W52.14 BOOL  ; 腔体下料#2夹爪气缸松开复位(M)
W52.15 BOOL  ; 腔体下料#3夹爪气缸夹紧复位(M)
W57.00 BOOL  ; 进料移栽有料信号
W60.00 BOOL  ; 腔体机构手复位
W60.01 BOOL  ; 腔体#1 & #2复位启动
W60.02 BOOL  ; 腔体#3 & #4复位启动
W61.01 BOOL  ; #1抽真空阀复位
W61.02 BOOL  ; #2抽真空阀复位
W61.03 BOOL  ; #1氦检阀复位
W61.04 BOOL  ; #2氦检阀复位
W61.05 BOOL  ; #1总氦检阀复位
W61.07 BOOL  ; #1合模气缸缩回位复位
W61.09 BOOL  ; #2合模气缸缩回位复位
W61.11 BOOL  ; 破真空阀#1&#2复位
W61.12 BOOL  ; 关破真空阀#1&#2复位
W61.15 BOOL  ; #1 & #2吹气阀复位
W62.00 BOOL  ; #2吹气阀复位
W62.01 BOOL  ; #3 & #4吹气阀复位
W62.03 BOOL  ; #3抽真空阀复位
W62.04 BOOL  ; #4抽真空阀复位
W62.06 BOOL  ; #2总氦检阀复位
W62.07 BOOL  ; 破真空阀#3&#4复位
W62.08 BOOL  ; 关破真空阀#3&#4复位
W62.09 BOOL  ; #3氦检阀复位
W62.10 BOOL  ; #4氦检阀复位
W62.11 BOOL  ; #3合模气缸缩回位复位
W62.12 BOOL  ; 破真空阀#3&#4复位
W62.13 BOOL  ; #4合模气缸缩回位复位
W70.00 BOOL  ; 出料机构手复位
W9.00 BOOL  ; 故障
W9.01 BOOL  ; 报警清除  HMI

## Program Main (cyclic task 0)
Local symbols
P_on BOOL

### Section 启停控制

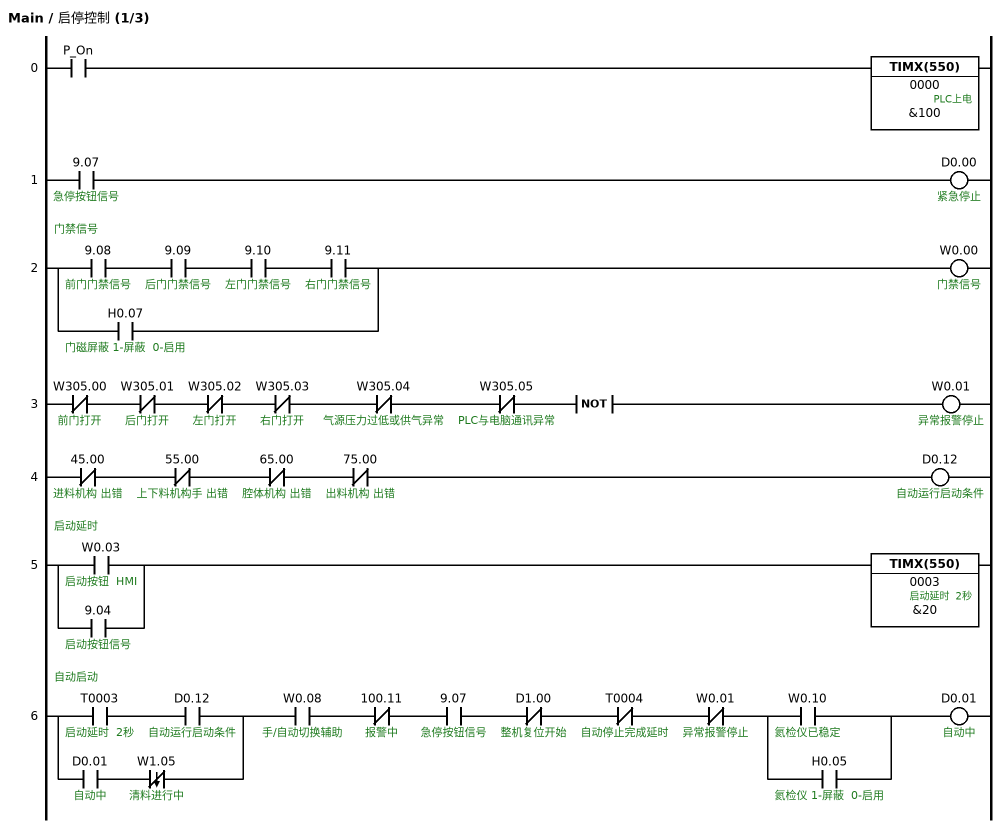
; rung 0
LD P_On
TIMX(550) 0000 &100  ; PLC上电
; rung 1
LD 9.07  ; 急停按钮信号
OUT D0.00  ; 紧急停止
; rung 2: 门禁信号
LD 9.08  ; 前门门禁信号
AND 9.09  ; 后门门禁信号
AND 9.10  ; 左门门禁信号
AND 9.11  ; 右门门禁信号
OR H0.07  ; 门磁屏蔽 1-屏蔽  0-启用
OUT W0.00  ; 门禁信号
; rung 3
LDNOT W305.00  ; 前门打开
ANDNOT W305.01  ; 后门打开
ANDNOT W305.02  ; 左门打开
ANDNOT W305.03  ; 右门打开
ANDNOT W305.04  ; 气源压力过低或供气异常
ANDNOT W305.05  ; PLC与电脑通讯异常
NOT(520)
OUT W0.01  ; 异常报警停止
; rung 4
LDNOT 45.00  ; 进料机构 出错
ANDNOT 55.00  ; 上下料机构手 出错
ANDNOT 65.00  ; 腔体机构 出错
ANDNOT 75.00  ; 出料机构 出错
OUT D0.12  ; 自动运行启动条件
; rung 5: 启动延时
LD W0.03  ; 启动按钮  HMI
OR 9.04  ; 启动按钮信号
TIMX(550) 0003 &20  ; 启动延时  2秒
; rung 6: 自动启动
LD T0003  ; 启动延时  2秒
AND D0.12  ; 自动运行启动条件
LD D0.01  ; 自动中
%ANDNOT W1.05  ; 清料进行中
ORLD
AND W0.08  ; 手/自动切换辅助
ANDNOT 100.11  ; 报警中
AND 9.07  ; 急停按钮信号
ANDNOT D1.00  ; 整机复位开始
ANDNOT T0004  ; 自动停止完成延时
ANDNOT W0.01  ; 异常报警停止
LD W0.10  ; 氦检仪已稳定
OR H0.05  ; 氦检仪 1-屏蔽  0-启用
ANDLD
OUT D0.01  ; 自动中

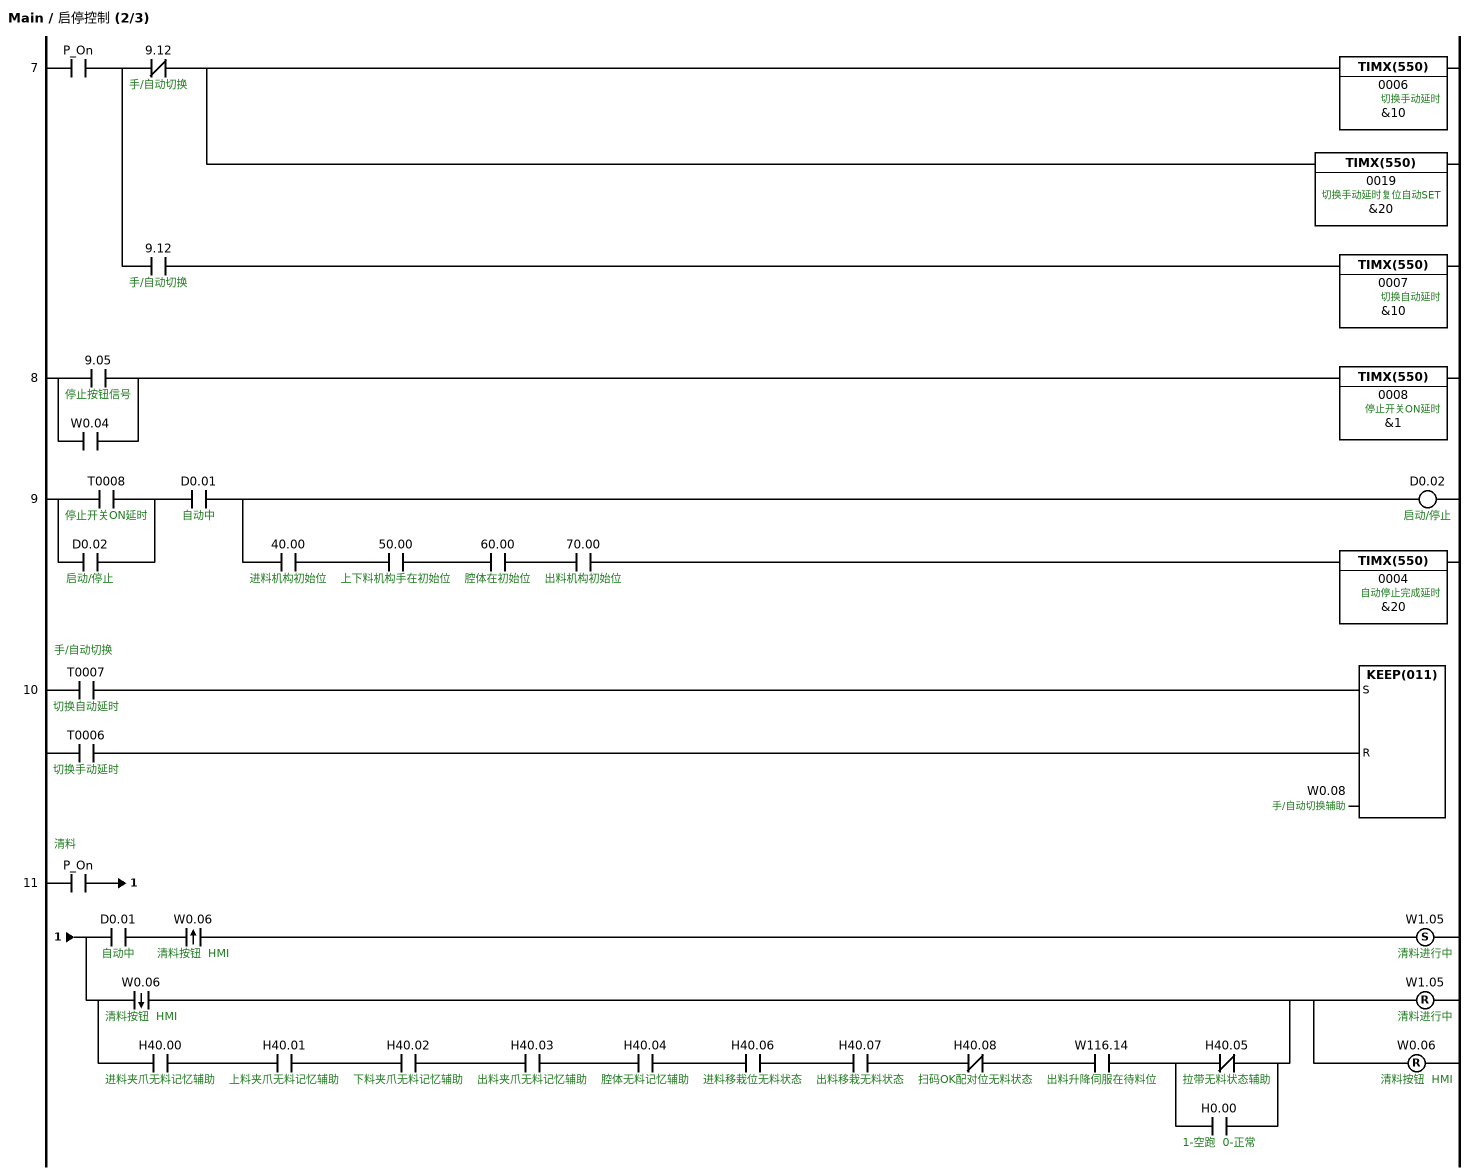
; rung 7
LD P_On
OUT TR0
ANDNOT 9.12  ; 手/自动切换
TIMX(550) 0006 &10  ; 切换手动延时
TIMX(550) 0019 &20  ; 切换手动延时复位自动SET
LD TR0
AND 9.12  ; 手/自动切换
TIMX(550) 0007 &10  ; 切换自动延时
; rung 8
LD 9.05  ; 停止按钮信号
OR W0.04
TIMX(550) 0008 &1  ; 停止开关ON延时
; rung 9
LD T0008  ; 停止开关ON延时
OR D0.02  ; 启动/停止
AND D0.01  ; 自动中
OUT D0.02  ; 启动/停止
AND 40.00  ; 进料机构初始位
AND 50.00  ; 上下料机构手在初始位
AND 60.00  ; 腔体在初始位
AND 70.00  ; 出料机构初始位
TIMX(550) 0004 &20  ; 自动停止完成延时
; rung 10: 手/自动切换
LD T0007  ; 切换自动延时
LD T0006  ; 切换手动延时
KEEP(011) W0.08  ; 手/自动切换辅助
; rung 11: 清料
LD P_On
OUT TR0
AND D0.01  ; 自动中
@AND W0.06  ; 清料按钮  HMI
SET W1.05  ; 清料进行中
LD TR0
%LD W0.06  ; 清料按钮  HMI
LD H40.00  ; 进料夹爪无料记忆辅助
AND H40.01  ; 上料夹爪无料记忆辅助
AND H40.02  ; 下料夹爪无料记忆辅助
AND H40.03  ; 出料夹爪无料记忆辅助
AND H40.04  ; 腔体无料记忆辅助
AND H40.06  ; 进料移栽位无料状态
AND H40.07  ; 出料移栽无料状态
ANDNOT H40.08  ; 扫码OK配对位无料状态
AND W116.14  ; 出料升降伺服在待料位
LDNOT H40.05  ; 拉带无料状态辅助
OR H0.00  ; 1-空跑  0-正常
ANDLD
ORLD
ANDLD
RSET W1.05  ; 清料进行中
RSET W0.06  ; 清料按钮  HMI

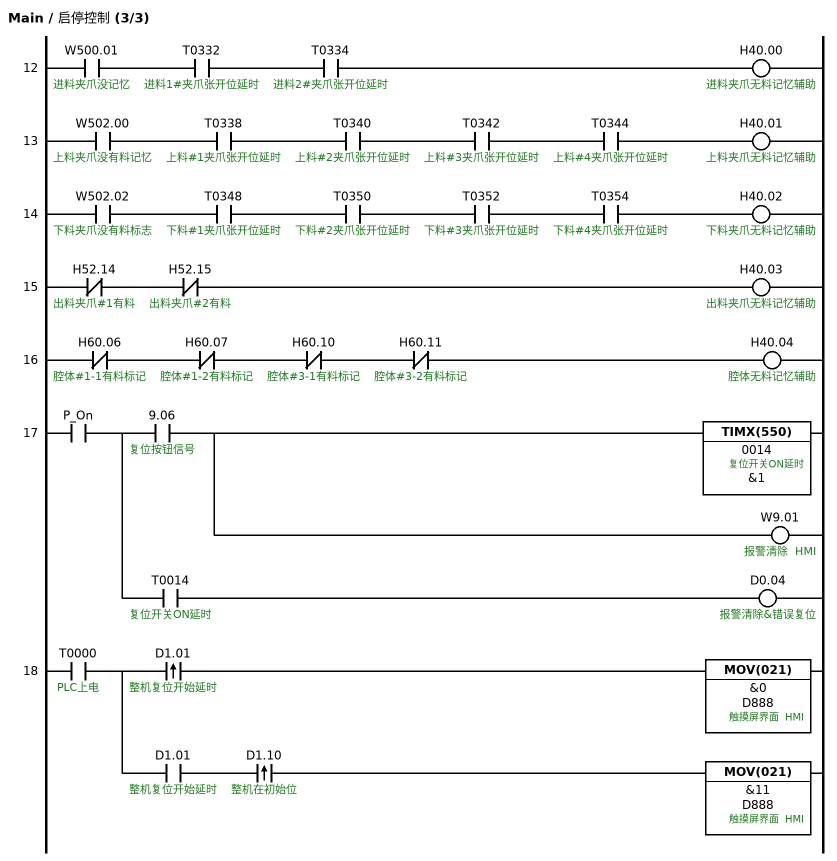
; rung 12
LD W500.01  ; 进料夹爪没记忆
AND T0332  ; 进料1#夹爪张开位延时
AND T0334  ; 进料2#夹爪张开位延时
OUT H40.00  ; 进料夹爪无料记忆辅助
; rung 13
LD W502.00  ; 上料夹爪没有料记忆
AND T0338  ; 上料#1夹爪张开位延时
AND T0340  ; 上料#2夹爪张开位延时
AND T0342  ; 上料#3夹爪张开位延时
AND T0344  ; 上料#4夹爪张开位延时
OUT H40.01  ; 上料夹爪无料记忆辅助
; rung 14
LD W502.02  ; 下料夹爪没有料标志
AND T0348  ; 下料#1夹爪张开位延时
AND T0350  ; 下料#2夹爪张开位延时
AND T0352  ; 下料#3夹爪张开位延时
AND T0354  ; 下料#4夹爪张开位延时
OUT H40.02  ; 下料夹爪无料记忆辅助
; rung 15
LDNOT H52.14  ; 出料夹爪#1有料
ANDNOT H52.15  ; 出料夹爪#2有料
OUT H40.03  ; 出料夹爪无料记忆辅助
; rung 16
LDNOT H60.06  ; 腔体#1-1有料标记
ANDNOT H60.07  ; 腔体#1-2有料标记
ANDNOT H60.10  ; 腔体#3-1有料标记
ANDNOT H60.11  ; 腔体#3-2有料标记
OUT H40.04  ; 腔体无料记忆辅助
; rung 17
LD P_On
OUT TR0
AND 9.06  ; 复位按钮信号
TIMX(550) 0014 &1  ; 复位开关ON延时
OUT W9.01  ; 报警清除  HMI
LD TR0
AND T0014  ; 复位开关ON延时
OUT D0.04  ; 报警清除&错误复位
; rung 18
LD T0000  ; PLC上电
OUT TR0
@AND D1.01  ; 整机复位开始延时
MOV(021) &0 D888  ; 触摸屏界面  HMI
LD TR0
AND D1.01  ; 整机复位开始延时
@AND D1.10  ; 整机在初始位
MOV(021) &11 D888  ; 触摸屏界面  HMI

### Section 传感器延时及屏蔽

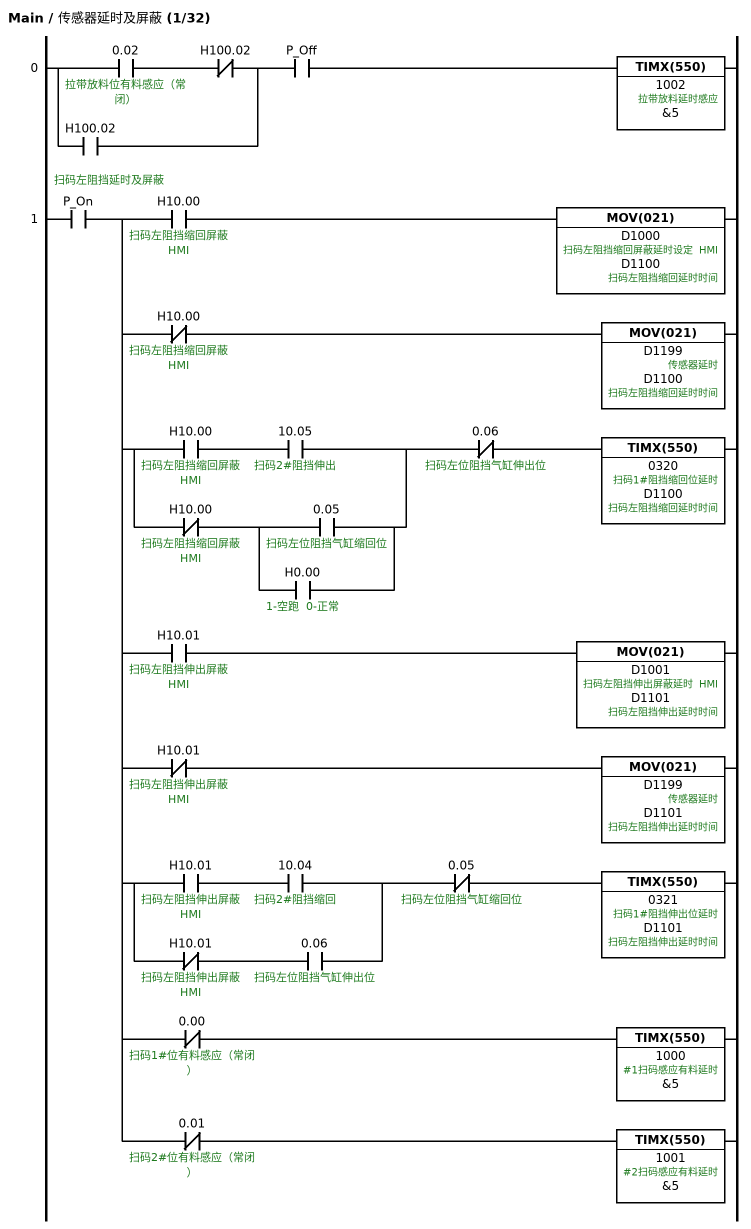
; rung 0
LD 0.02  ; 拉带放料位有料感应（常闭）
ANDNOT H100.02
OR H100.02
AND P_Off
TIMX(550) 1002 &5  ; 拉带放料延时感应
; rung 1: 扫码左阻挡延时及屏蔽
LD P_On
OUT TR0
AND H10.00  ; 扫码左阻挡缩回屏蔽  HMI
MOV(021) D1000 D1100  ; 扫码左阻挡缩回屏蔽延时设定  HMI, 扫码左阻挡缩回延时时间
LD TR0
ANDNOT H10.00  ; 扫码左阻挡缩回屏蔽  HMI
MOV(021) D1199 D1100  ; 传感器延时, 扫码左阻挡缩回延时时间
LD TR0
LD H10.00  ; 扫码左阻挡缩回屏蔽  HMI
AND 10.05  ; 扫码2#阻挡伸出
LDNOT H10.00  ; 扫码左阻挡缩回屏蔽  HMI
LD 0.05  ; 扫码左位阻挡气缸缩回位
OR H0.00  ; 1-空跑  0-正常
ANDLD
ORLD
ANDLD
ANDNOT 0.06  ; 扫码左位阻挡气缸伸出位
TIMX(550) 0320 D1100  ; 扫码左阻挡缩回延时时间, 扫码1#阻挡缩回位延时
LD TR0
AND H10.01  ; 扫码左阻挡伸出屏蔽  HMI
MOV(021) D1001 D1101  ; 扫码左阻挡伸出屏蔽延时  HMI, 扫码左阻挡伸出延时时间
LD TR0
ANDNOT H10.01  ; 扫码左阻挡伸出屏蔽  HMI
MOV(021) D1199 D1101  ; 传感器延时, 扫码左阻挡伸出延时时间
LD TR0
LD H10.01  ; 扫码左阻挡伸出屏蔽  HMI
AND 10.04  ; 扫码2#阻挡缩回
LDNOT H10.01  ; 扫码左阻挡伸出屏蔽  HMI
AND 0.06  ; 扫码左位阻挡气缸伸出位
ORLD
ANDLD
ANDNOT 0.05  ; 扫码左位阻挡气缸缩回位
TIMX(550) 0321 D1101  ; 扫码左阻挡伸出延时时间, 扫码1#阻挡伸出位延时
LD TR0
ANDNOT 0.00  ; 扫码1#位有料感应（常闭）
TIMX(550) 1000 &5  ; #1扫码感应有料延时
LD TR0
ANDNOT 0.01  ; 扫码2#位有料感应（常闭）
TIMX(550) 1001 &5  ; #2扫码感应有料延时

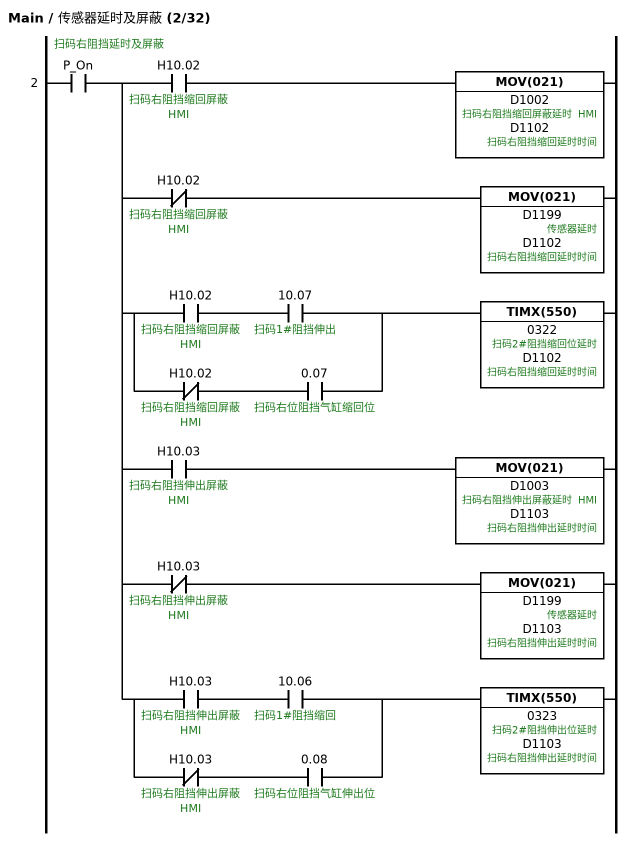
; rung 2: 扫码右阻挡延时及屏蔽
LD P_On
OUT TR0
AND H10.02  ; 扫码右阻挡缩回屏蔽  HMI
MOV(021) D1002 D1102  ; 扫码右阻挡缩回屏蔽延时  HMI, 扫码右阻挡缩回延时时间
LD TR0
ANDNOT H10.02  ; 扫码右阻挡缩回屏蔽  HMI
MOV(021) D1199 D1102  ; 传感器延时, 扫码右阻挡缩回延时时间
LD TR0
LD H10.02  ; 扫码右阻挡缩回屏蔽  HMI
AND 10.07  ; 扫码1#阻挡伸出
LDNOT H10.02  ; 扫码右阻挡缩回屏蔽  HMI
AND 0.07  ; 扫码右位阻挡气缸缩回位
ORLD
ANDLD
TIMX(550) 0322 D1102  ; 扫码右阻挡缩回延时时间, 扫码2#阻挡缩回位延时
LD TR0
AND H10.03  ; 扫码右阻挡伸出屏蔽  HMI
MOV(021) D1003 D1103  ; 扫码右阻挡伸出屏蔽延时  HMI, 扫码右阻挡伸出延时时间
LD TR0
ANDNOT H10.03  ; 扫码右阻挡伸出屏蔽  HMI
MOV(021) D1199 D1103  ; 传感器延时, 扫码右阻挡伸出延时时间
LD TR0
LD H10.03  ; 扫码右阻挡伸出屏蔽  HMI
AND 10.06  ; 扫码1#阻挡缩回
LDNOT H10.03  ; 扫码右阻挡伸出屏蔽  HMI
AND 0.08  ; 扫码右位阻挡气缸伸出位
ORLD
ANDLD
TIMX(550) 0323 D1103  ; 扫码右阻挡伸出延时时间, 扫码2#阻挡伸出位延时

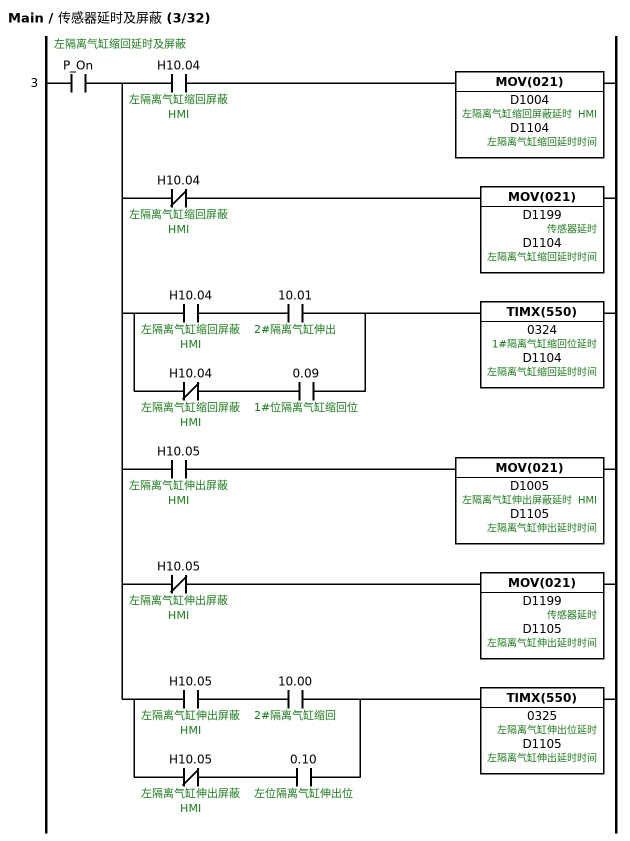
; rung 3: 左隔离气缸缩回延时及屏蔽
LD P_On
OUT TR0
AND H10.04  ; 左隔离气缸缩回屏蔽  HMI
MOV(021) D1004 D1104  ; 左隔离气缸缩回屏蔽延时  HMI, 左隔离气缸缩回延时时间
LD TR0
ANDNOT H10.04  ; 左隔离气缸缩回屏蔽  HMI
MOV(021) D1199 D1104  ; 传感器延时, 左隔离气缸缩回延时时间
LD TR0
LD H10.04  ; 左隔离气缸缩回屏蔽  HMI
AND 10.01  ; 2#隔离气缸伸出
LDNOT H10.04  ; 左隔离气缸缩回屏蔽  HMI
AND 0.09  ; 1#位隔离气缸缩回位
ORLD
ANDLD
TIMX(550) 0324 D1104  ; 左隔离气缸缩回延时时间, 1#隔离气缸缩回位延时
LD TR0
AND H10.05  ; 左隔离气缸伸出屏蔽  HMI
MOV(021) D1005 D1105  ; 左隔离气缸伸出屏蔽延时  HMI, 左隔离气缸伸出延时时间
LD TR0
ANDNOT H10.05  ; 左隔离气缸伸出屏蔽  HMI
MOV(021) D1199 D1105  ; 传感器延时, 左隔离气缸伸出延时时间
LD TR0
LD H10.05  ; 左隔离气缸伸出屏蔽  HMI
AND 10.00  ; 2#隔离气缸缩回
LDNOT H10.05  ; 左隔离气缸伸出屏蔽  HMI
AND 0.10  ; 左位隔离气缸伸出位
ORLD
ANDLD
TIMX(550) 0325 D1105  ; 左隔离气缸伸出延时时间, 左隔离气缸伸出位延时

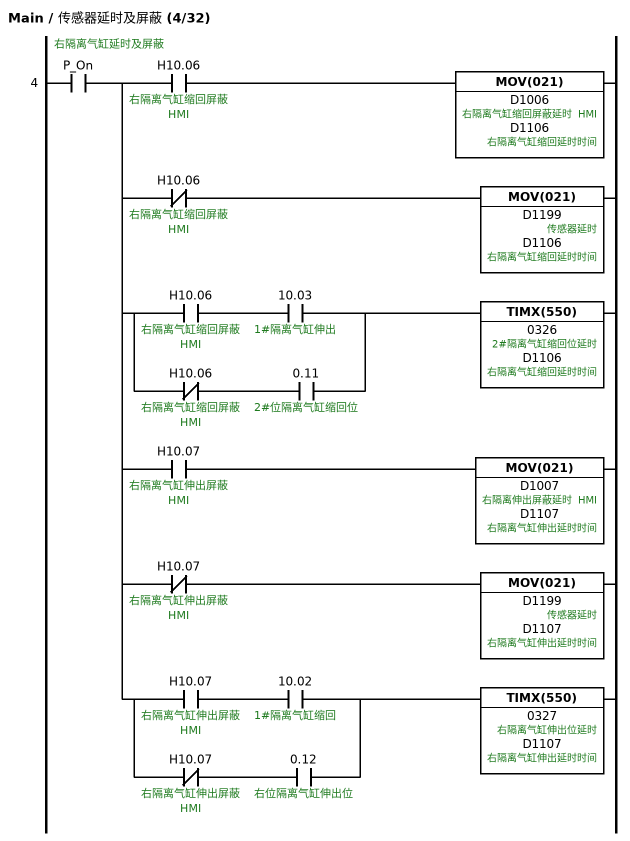
; rung 4: 右隔离气缸延时及屏蔽
LD P_On
OUT TR0
AND H10.06  ; 右隔离气缸缩回屏蔽  HMI
MOV(021) D1006 D1106  ; 右隔离气缸缩回屏蔽延时  HMI, 右隔离气缸缩回延时时间
LD TR0
ANDNOT H10.06  ; 右隔离气缸缩回屏蔽  HMI
MOV(021) D1199 D1106  ; 传感器延时, 右隔离气缸缩回延时时间
LD TR0
LD H10.06  ; 右隔离气缸缩回屏蔽  HMI
AND 10.03  ; 1#隔离气缸伸出
LDNOT H10.06  ; 右隔离气缸缩回屏蔽  HMI
AND 0.11  ; 2#位隔离气缸缩回位
ORLD
ANDLD
TIMX(550) 0326 D1106  ; 右隔离气缸缩回延时时间, 2#隔离气缸缩回位延时
LD TR0
AND H10.07  ; 右隔离气缸伸出屏蔽  HMI
MOV(021) D1007 D1107  ; 右隔离伸出屏蔽延时  HMI, 右隔离气缸伸出延时时间
LD TR0
ANDNOT H10.07  ; 右隔离气缸伸出屏蔽  HMI
MOV(021) D1199 D1107  ; 传感器延时, 右隔离气缸伸出延时时间
LD TR0
LD H10.07  ; 右隔离气缸伸出屏蔽  HMI
AND 10.02  ; 1#隔离气缸缩回
LDNOT H10.07  ; 右隔离气缸伸出屏蔽  HMI
AND 0.12  ; 右位隔离气缸伸出位
ORLD
ANDLD
TIMX(550) 0327 D1107  ; 右隔离气缸伸出延时时间, 右隔离气缸伸出位延时

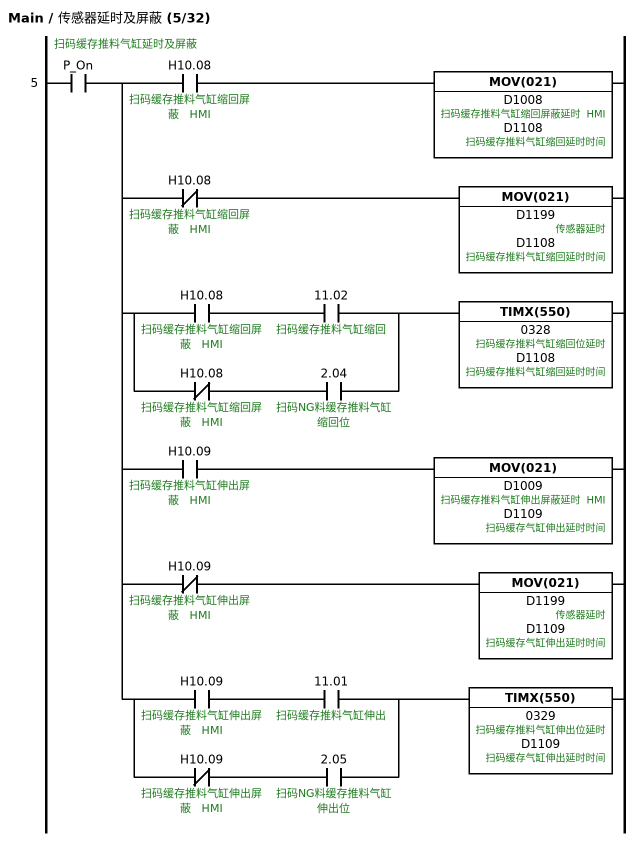
; rung 5: 扫码缓存推料气缸延时及屏蔽
LD P_On
OUT TR0
AND H10.08  ; 扫码缓存推料气缸缩回屏蔽   HMI
MOV(021) D1008 D1108  ; 扫码缓存推料气缸缩回屏蔽延时  HMI, 扫码缓存推料气缸缩回延时时间
LD TR0
ANDNOT H10.08  ; 扫码缓存推料气缸缩回屏蔽   HMI
MOV(021) D1199 D1108  ; 传感器延时, 扫码缓存推料气缸缩回延时时间
LD TR0
LD H10.08  ; 扫码缓存推料气缸缩回屏蔽   HMI
AND 11.02  ; 扫码缓存推料气缸缩回
LDNOT H10.08  ; 扫码缓存推料气缸缩回屏蔽   HMI
AND 2.04  ; 扫码NG料缓存推料气缸缩回位
ORLD
ANDLD
TIMX(550) 0328 D1108  ; 扫码缓存推料气缸缩回延时时间, 扫码缓存推料气缸缩回位延时
LD TR0
AND H10.09  ; 扫码缓存推料气缸伸出屏蔽   HMI
MOV(021) D1009 D1109  ; 扫码缓存推料气缸伸出屏蔽延时  HMI, 扫码缓存气缸伸出延时时间
LD TR0
ANDNOT H10.09  ; 扫码缓存推料气缸伸出屏蔽   HMI
MOV(021) D1199 D1109  ; 传感器延时, 扫码缓存气缸伸出延时时间
LD TR0
LD H10.09  ; 扫码缓存推料气缸伸出屏蔽   HMI
AND 11.01  ; 扫码缓存推料气缸伸出
LDNOT H10.09  ; 扫码缓存推料气缸伸出屏蔽   HMI
AND 2.05  ; 扫码NG料缓存推料气缸伸出位
ORLD
ANDLD
TIMX(550) 0329 D1109  ; 扫码缓存气缸伸出延时时间, 扫码缓存推料气缸伸出位延时

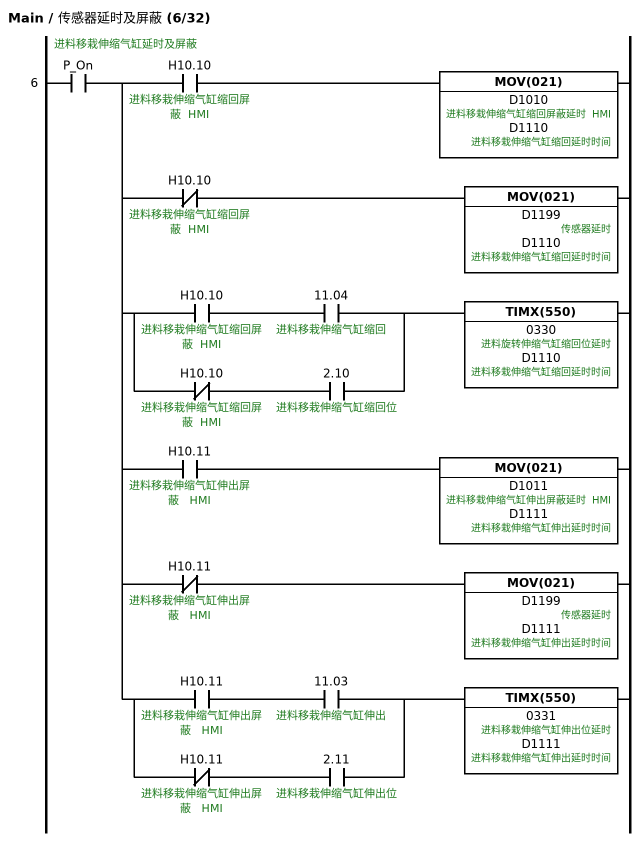
; rung 6: 进料移栽伸缩气缸延时及屏蔽
LD P_On
OUT TR0
AND H10.10  ; 进料移栽伸缩气缸缩回屏蔽  HMI
MOV(021) D1010 D1110  ; 进料移栽伸缩气缸缩回屏蔽延时  HMI, 进料移栽伸缩气缸缩回延时时间
LD TR0
ANDNOT H10.10  ; 进料移栽伸缩气缸缩回屏蔽  HMI
MOV(021) D1199 D1110  ; 传感器延时, 进料移栽伸缩气缸缩回延时时间
LD TR0
LD H10.10  ; 进料移栽伸缩气缸缩回屏蔽  HMI
AND 11.04  ; 进料移栽伸缩气缸缩回
LDNOT H10.10  ; 进料移栽伸缩气缸缩回屏蔽  HMI
AND 2.10  ; 进料移栽伸缩气缸缩回位
ORLD
ANDLD
TIMX(550) 0330 D1110  ; 进料移栽伸缩气缸缩回延时时间, 进料旋转伸缩气缸缩回位延时
LD TR0
AND H10.11  ; 进料移栽伸缩气缸伸出屏蔽   HMI
MOV(021) D1011 D1111  ; 进料移栽伸缩气缸伸出屏蔽延时  HMI, 进料移栽伸缩气缸伸出延时时间
LD TR0
ANDNOT H10.11  ; 进料移栽伸缩气缸伸出屏蔽   HMI
MOV(021) D1199 D1111  ; 传感器延时, 进料移栽伸缩气缸伸出延时时间
LD TR0
LD H10.11  ; 进料移栽伸缩气缸伸出屏蔽   HMI
AND 11.03  ; 进料移栽伸缩气缸伸出
LDNOT H10.11  ; 进料移栽伸缩气缸伸出屏蔽   HMI
AND 2.11  ; 进料移栽伸缩气缸伸出位
ORLD
ANDLD
TIMX(550) 0331 D1111  ; 进料移栽伸缩气缸伸出延时时间, 进料移栽伸缩气缸伸出位延时

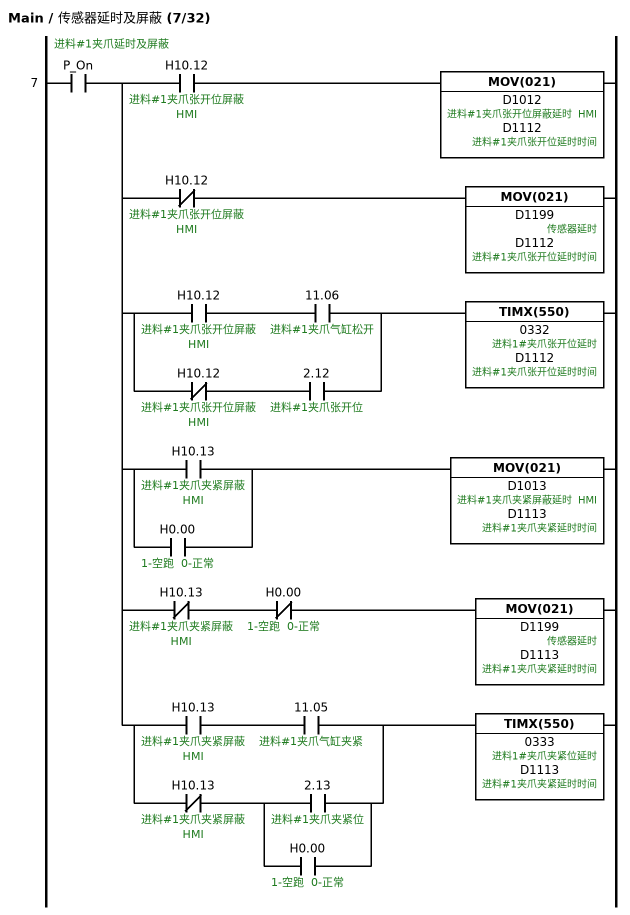
; rung 7: 进料#1夹爪延时及屏蔽
LD P_On
OUT TR0
AND H10.12  ; 进料#1夹爪张开位屏蔽  HMI
MOV(021) D1012 D1112  ; 进料#1夹爪张开位屏蔽延时  HMI, 进料#1夹爪张开位延时时间
LD TR0
ANDNOT H10.12  ; 进料#1夹爪张开位屏蔽  HMI
MOV(021) D1199 D1112  ; 传感器延时, 进料#1夹爪张开位延时时间
LD TR0
LD H10.12  ; 进料#1夹爪张开位屏蔽  HMI
AND 11.06  ; 进料#1夹爪气缸松开
LDNOT H10.12  ; 进料#1夹爪张开位屏蔽  HMI
AND 2.12  ; 进料#1夹爪张开位
ORLD
ANDLD
TIMX(550) 0332 D1112  ; 进料#1夹爪张开位延时时间, 进料1#夹爪张开位延时
LD TR0
LD H10.13  ; 进料#1夹爪夹紧屏蔽  HMI
OR H0.00  ; 1-空跑  0-正常
ANDLD
MOV(021) D1013 D1113  ; 进料#1夹爪夹紧屏蔽延时  HMI, 进料#1夹爪夹紧延时时间
LD TR0
ANDNOT H10.13  ; 进料#1夹爪夹紧屏蔽  HMI
ANDNOT H0.00  ; 1-空跑  0-正常
MOV(021) D1199 D1113  ; 传感器延时, 进料#1夹爪夹紧延时时间
LD TR0
LD H10.13  ; 进料#1夹爪夹紧屏蔽  HMI
AND 11.05  ; 进料#1夹爪气缸夹紧
LDNOT H10.13  ; 进料#1夹爪夹紧屏蔽  HMI
LD 2.13  ; 进料#1夹爪夹紧位
OR H0.00  ; 1-空跑  0-正常
ANDLD
ORLD
ANDLD
TIMX(550) 0333 D1113  ; 进料#1夹爪夹紧延时时间, 进料1#夹爪夹紧位延时

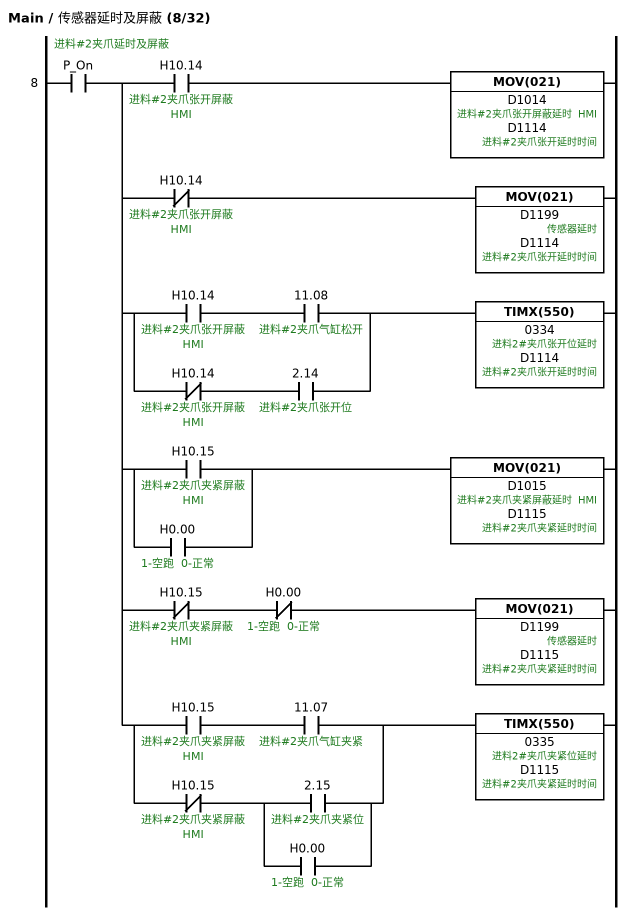
; rung 8: 进料#2夹爪延时及屏蔽
LD P_On
OUT TR0
AND H10.14  ; 进料#2夹爪张开屏蔽  HMI
MOV(021) D1014 D1114  ; 进料#2夹爪张开屏蔽延时  HMI, 进料#2夹爪张开延时时间
LD TR0
ANDNOT H10.14  ; 进料#2夹爪张开屏蔽  HMI
MOV(021) D1199 D1114  ; 传感器延时, 进料#2夹爪张开延时时间
LD TR0
LD H10.14  ; 进料#2夹爪张开屏蔽  HMI
AND 11.08  ; 进料#2夹爪气缸松开
LDNOT H10.14  ; 进料#2夹爪张开屏蔽  HMI
AND 2.14  ; 进料#2夹爪张开位
ORLD
ANDLD
TIMX(550) 0334 D1114  ; 进料#2夹爪张开延时时间, 进料2#夹爪张开位延时
LD TR0
LD H10.15  ; 进料#2夹爪夹紧屏蔽  HMI
OR H0.00  ; 1-空跑  0-正常
ANDLD
MOV(021) D1015 D1115  ; 进料#2夹爪夹紧屏蔽延时  HMI, 进料#2夹爪夹紧延时时间
LD TR0
ANDNOT H10.15  ; 进料#2夹爪夹紧屏蔽  HMI
ANDNOT H0.00  ; 1-空跑  0-正常
MOV(021) D1199 D1115  ; 传感器延时, 进料#2夹爪夹紧延时时间
LD TR0
LD H10.15  ; 进料#2夹爪夹紧屏蔽  HMI
AND 11.07  ; 进料#2夹爪气缸夹紧
LDNOT H10.15  ; 进料#2夹爪夹紧屏蔽  HMI
LD 2.15  ; 进料#2夹爪夹紧位
OR H0.00  ; 1-空跑  0-正常
ANDLD
ORLD
ANDLD
TIMX(550) 0335 D1115  ; 进料#2夹爪夹紧延时时间, 进料2#夹爪夹紧位延时

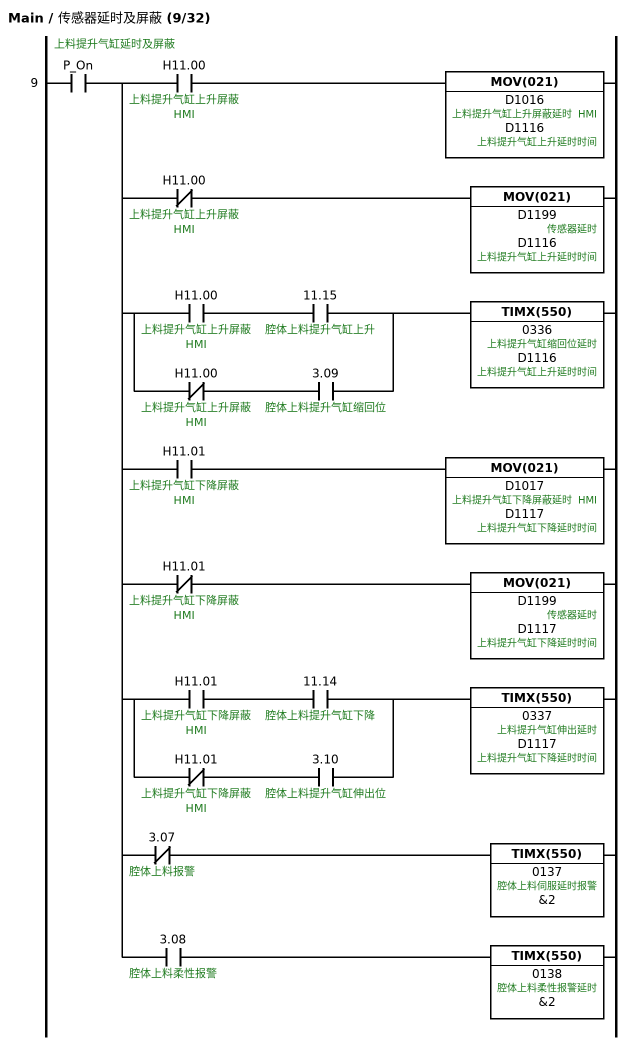
; rung 9: 上料提升气缸延时及屏蔽
LD P_On
OUT TR0
AND H11.00  ; 上料提升气缸上升屏蔽  HMI
MOV(021) D1016 D1116  ; 上料提升气缸上升屏蔽延时  HMI, 上料提升气缸上升延时时间
LD TR0
ANDNOT H11.00  ; 上料提升气缸上升屏蔽  HMI
MOV(021) D1199 D1116  ; 传感器延时, 上料提升气缸上升延时时间
LD TR0
LD H11.00  ; 上料提升气缸上升屏蔽  HMI
AND 11.15  ; 腔体上料提升气缸上升
LDNOT H11.00  ; 上料提升气缸上升屏蔽  HMI
AND 3.09  ; 腔体上料提升气缸缩回位
ORLD
ANDLD
TIMX(550) 0336 D1116  ; 上料提升气缸上升延时时间, 上料提升气缸缩回位延时
LD TR0
AND H11.01  ; 上料提升气缸下降屏蔽  HMI
MOV(021) D1017 D1117  ; 上料提升气缸下降屏蔽延时  HMI, 上料提升气缸下降延时时间
LD TR0
ANDNOT H11.01  ; 上料提升气缸下降屏蔽  HMI
MOV(021) D1199 D1117  ; 传感器延时, 上料提升气缸下降延时时间
LD TR0
LD H11.01  ; 上料提升气缸下降屏蔽  HMI
AND 11.14  ; 腔体上料提升气缸下降
LDNOT H11.01  ; 上料提升气缸下降屏蔽  HMI
AND 3.10  ; 腔体上料提升气缸伸出位
ORLD
ANDLD
TIMX(550) 0337 D1117  ; 上料提升气缸下降延时时间, 上料提升气缸伸出延时
LD TR0
ANDNOT 3.07  ; 腔体上料报警
TIMX(550) 0137 &2  ; 腔体上料伺服延时报警
LD TR0
AND 3.08  ; 腔体上料柔性报警
TIMX(550) 0138 &2  ; 腔体上料柔性报警延时

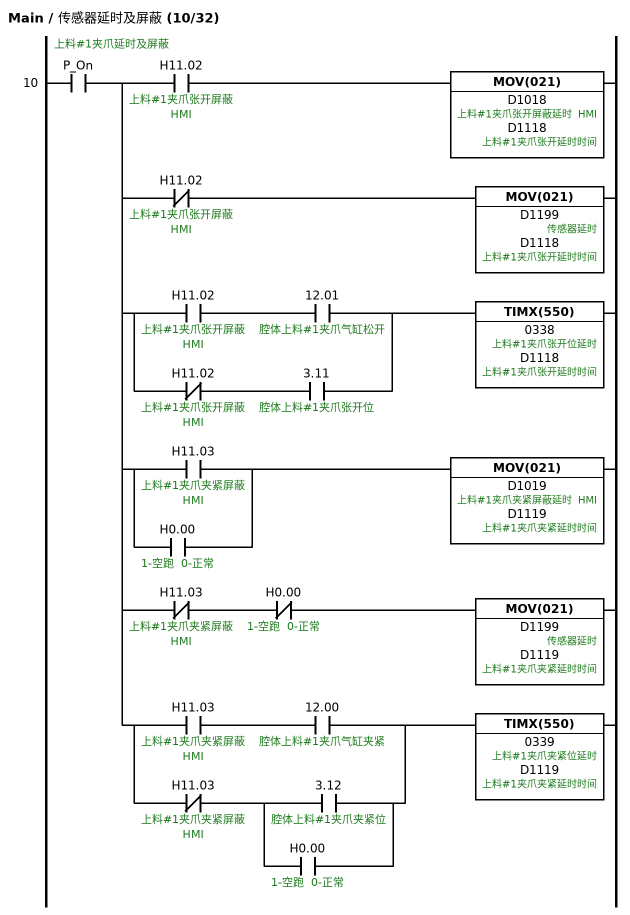
; rung 10: 上料#1夹爪延时及屏蔽
LD P_On
OUT TR0
AND H11.02  ; 上料#1夹爪张开屏蔽  HMI
MOV(021) D1018 D1118  ; 上料#1夹爪张开屏蔽延时  HMI, 上料#1夹爪张开延时时间
LD TR0
ANDNOT H11.02  ; 上料#1夹爪张开屏蔽  HMI
MOV(021) D1199 D1118  ; 传感器延时, 上料#1夹爪张开延时时间
LD TR0
LD H11.02  ; 上料#1夹爪张开屏蔽  HMI
AND 12.01  ; 腔体上料#1夹爪气缸松开
LDNOT H11.02  ; 上料#1夹爪张开屏蔽  HMI
AND 3.11  ; 腔体上料#1夹爪张开位
ORLD
ANDLD
TIMX(550) 0338 D1118  ; 上料#1夹爪张开延时时间, 上料#1夹爪张开位延时
LD TR0
LD H11.03  ; 上料#1夹爪夹紧屏蔽  HMI
OR H0.00  ; 1-空跑  0-正常
ANDLD
MOV(021) D1019 D1119  ; 上料#1夹爪夹紧屏蔽延时  HMI, 上料#1夹爪夹紧延时时间
LD TR0
ANDNOT H11.03  ; 上料#1夹爪夹紧屏蔽  HMI
ANDNOT H0.00  ; 1-空跑  0-正常
MOV(021) D1199 D1119  ; 传感器延时, 上料#1夹爪夹紧延时时间
LD TR0
LD H11.03  ; 上料#1夹爪夹紧屏蔽  HMI
AND 12.00  ; 腔体上料#1夹爪气缸夹紧
LDNOT H11.03  ; 上料#1夹爪夹紧屏蔽  HMI
LD 3.12  ; 腔体上料#1夹爪夹紧位
OR H0.00  ; 1-空跑  0-正常
ANDLD
ORLD
ANDLD
TIMX(550) 0339 D1119  ; 上料#1夹爪夹紧延时时间, 上料#1夹爪夹紧位延时

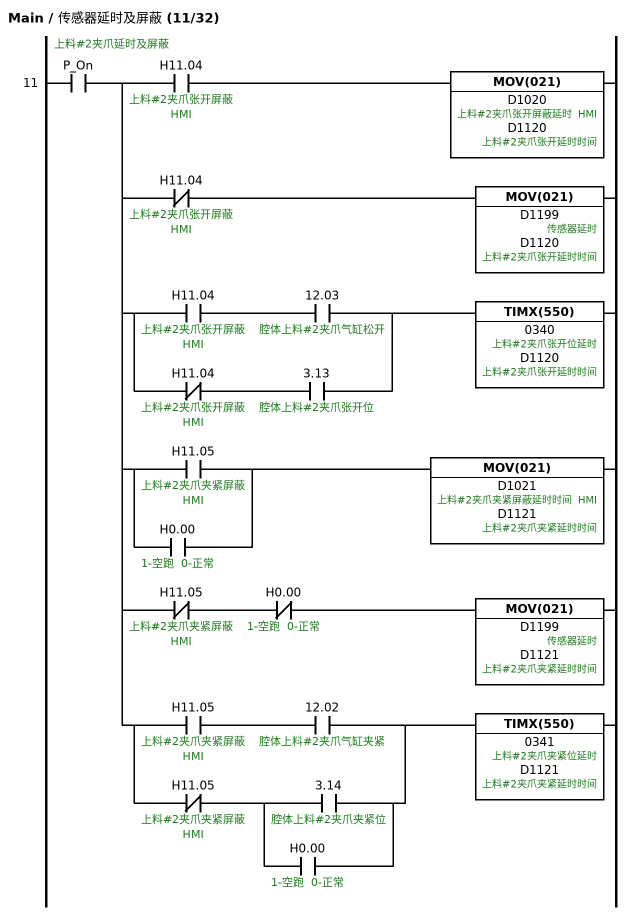
; rung 11: 上料#2夹爪延时及屏蔽
LD P_On
OUT TR0
AND H11.04  ; 上料#2夹爪张开屏蔽  HMI
MOV(021) D1020 D1120  ; 上料#2夹爪张开屏蔽延时  HMI, 上料#2夹爪张开延时时间
LD TR0
ANDNOT H11.04  ; 上料#2夹爪张开屏蔽  HMI
MOV(021) D1199 D1120  ; 传感器延时, 上料#2夹爪张开延时时间
LD TR0
LD H11.04  ; 上料#2夹爪张开屏蔽  HMI
AND 12.03  ; 腔体上料#2夹爪气缸松开
LDNOT H11.04  ; 上料#2夹爪张开屏蔽  HMI
AND 3.13  ; 腔体上料#2夹爪张开位
ORLD
ANDLD
TIMX(550) 0340 D1120  ; 上料#2夹爪张开延时时间, 上料#2夹爪张开位延时
LD TR0
LD H11.05  ; 上料#2夹爪夹紧屏蔽  HMI
OR H0.00  ; 1-空跑  0-正常
ANDLD
MOV(021) D1021 D1121  ; 上料#2夹爪夹紧屏蔽延时时间  HMI, 上料#2夹爪夹紧延时时间
LD TR0
ANDNOT H11.05  ; 上料#2夹爪夹紧屏蔽  HMI
ANDNOT H0.00  ; 1-空跑  0-正常
MOV(021) D1199 D1121  ; 传感器延时, 上料#2夹爪夹紧延时时间
LD TR0
LD H11.05  ; 上料#2夹爪夹紧屏蔽  HMI
AND 12.02  ; 腔体上料#2夹爪气缸夹紧
LDNOT H11.05  ; 上料#2夹爪夹紧屏蔽  HMI
LD 3.14  ; 腔体上料#2夹爪夹紧位
OR H0.00  ; 1-空跑  0-正常
ANDLD
ORLD
ANDLD
TIMX(550) 0341 D1121  ; 上料#2夹爪夹紧延时时间, 上料#2夹爪夹紧位延时

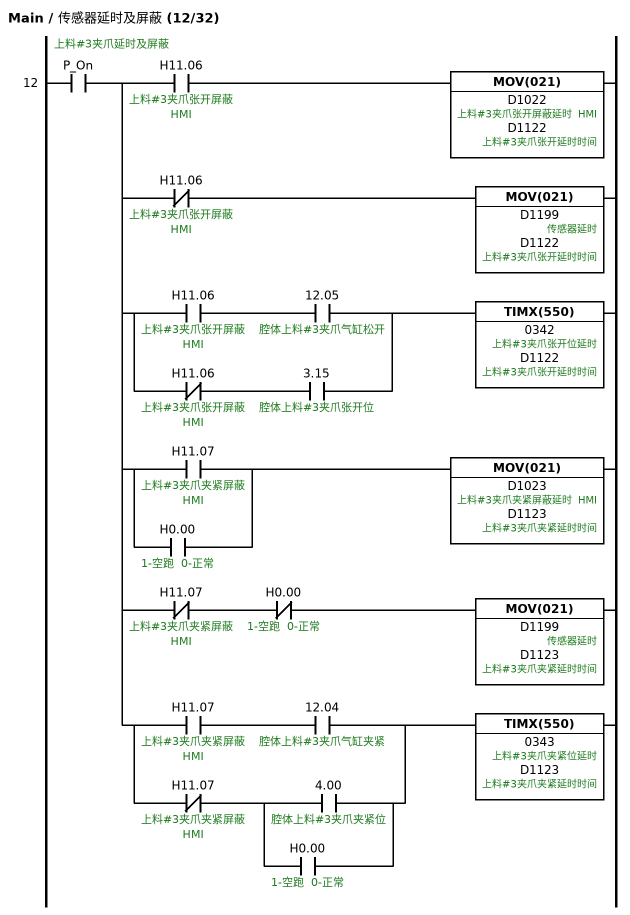
; rung 12: 上料#3夹爪延时及屏蔽
LD P_On
OUT TR0
AND H11.06  ; 上料#3夹爪张开屏蔽  HMI
MOV(021) D1022 D1122  ; 上料#3夹爪张开屏蔽延时  HMI, 上料#3夹爪张开延时时间
LD TR0
ANDNOT H11.06  ; 上料#3夹爪张开屏蔽  HMI
MOV(021) D1199 D1122  ; 传感器延时, 上料#3夹爪张开延时时间
LD TR0
LD H11.06  ; 上料#3夹爪张开屏蔽  HMI
AND 12.05  ; 腔体上料#3夹爪气缸松开
LDNOT H11.06  ; 上料#3夹爪张开屏蔽  HMI
AND 3.15  ; 腔体上料#3夹爪张开位
ORLD
ANDLD
TIMX(550) 0342 D1122  ; 上料#3夹爪张开延时时间, 上料#3夹爪张开位延时
LD TR0
LD H11.07  ; 上料#3夹爪夹紧屏蔽  HMI
OR H0.00  ; 1-空跑  0-正常
ANDLD
MOV(021) D1023 D1123  ; 上料#3夹爪夹紧屏蔽延时  HMI, 上料#3夹爪夹紧延时时间
LD TR0
ANDNOT H11.07  ; 上料#3夹爪夹紧屏蔽  HMI
ANDNOT H0.00  ; 1-空跑  0-正常
MOV(021) D1199 D1123  ; 传感器延时, 上料#3夹爪夹紧延时时间
LD TR0
LD H11.07  ; 上料#3夹爪夹紧屏蔽  HMI
AND 12.04  ; 腔体上料#3夹爪气缸夹紧
LDNOT H11.07  ; 上料#3夹爪夹紧屏蔽  HMI
LD 4.00  ; 腔体上料#3夹爪夹紧位
OR H0.00  ; 1-空跑  0-正常
ANDLD
ORLD
ANDLD
TIMX(550) 0343 D1123  ; 上料#3夹爪夹紧延时时间, 上料#3夹爪夹紧位延时

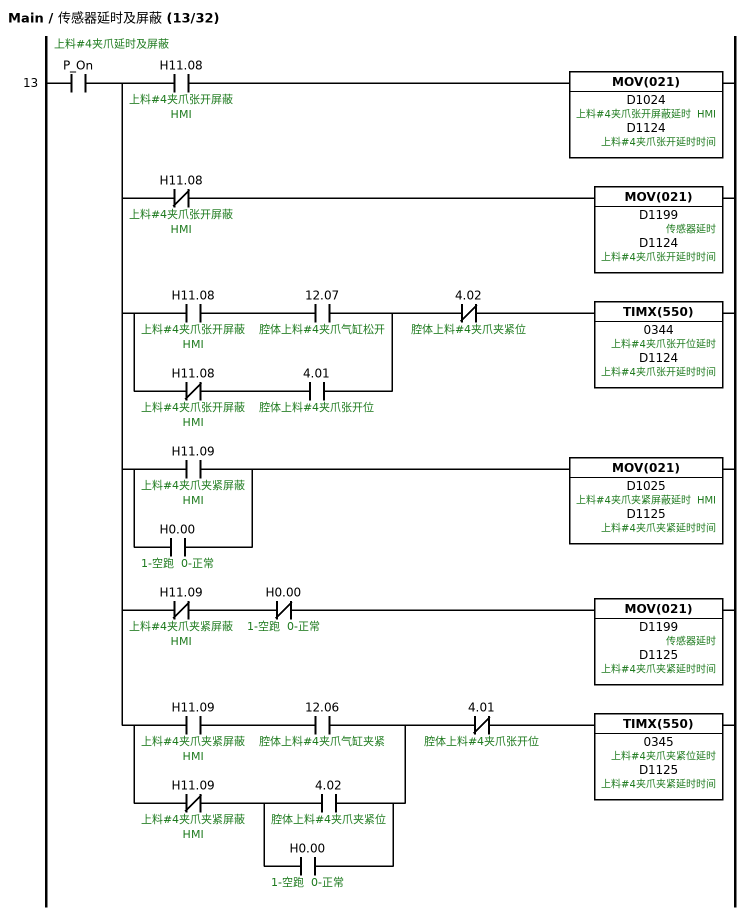
; rung 13: 上料#4夹爪延时及屏蔽
LD P_On
OUT TR0
AND H11.08  ; 上料#4夹爪张开屏蔽  HMI
MOV(021) D1024 D1124  ; 上料#4夹爪张开屏蔽延时  HMI, 上料#4夹爪张开延时时间
LD TR0
ANDNOT H11.08  ; 上料#4夹爪张开屏蔽  HMI
MOV(021) D1199 D1124  ; 传感器延时, 上料#4夹爪张开延时时间
LD TR0
LD H11.08  ; 上料#4夹爪张开屏蔽  HMI
AND 12.07  ; 腔体上料#4夹爪气缸松开
LDNOT H11.08  ; 上料#4夹爪张开屏蔽  HMI
AND 4.01  ; 腔体上料#4夹爪张开位
ORLD
ANDLD
ANDNOT 4.02  ; 腔体上料#4夹爪夹紧位
TIMX(550) 0344 D1124  ; 上料#4夹爪张开延时时间, 上料#4夹爪张开位延时
LD TR0
LD H11.09  ; 上料#4夹爪夹紧屏蔽  HMI
OR H0.00  ; 1-空跑  0-正常
ANDLD
MOV(021) D1025 D1125  ; 上料#4夹爪夹紧屏蔽延时  HMI, 上料#4夹爪夹紧延时时间
LD TR0
ANDNOT H11.09  ; 上料#4夹爪夹紧屏蔽  HMI
ANDNOT H0.00  ; 1-空跑  0-正常
MOV(021) D1199 D1125  ; 传感器延时, 上料#4夹爪夹紧延时时间
LD TR0
LD H11.09  ; 上料#4夹爪夹紧屏蔽  HMI
AND 12.06  ; 腔体上料#4夹爪气缸夹紧
LDNOT H11.09  ; 上料#4夹爪夹紧屏蔽  HMI
LD 4.02  ; 腔体上料#4夹爪夹紧位
OR H0.00  ; 1-空跑  0-正常
ANDLD
ORLD
ANDLD
ANDNOT 4.01  ; 腔体上料#4夹爪张开位
TIMX(550) 0345 D1125  ; 上料#4夹爪夹紧延时时间, 上料#4夹爪夹紧位延时

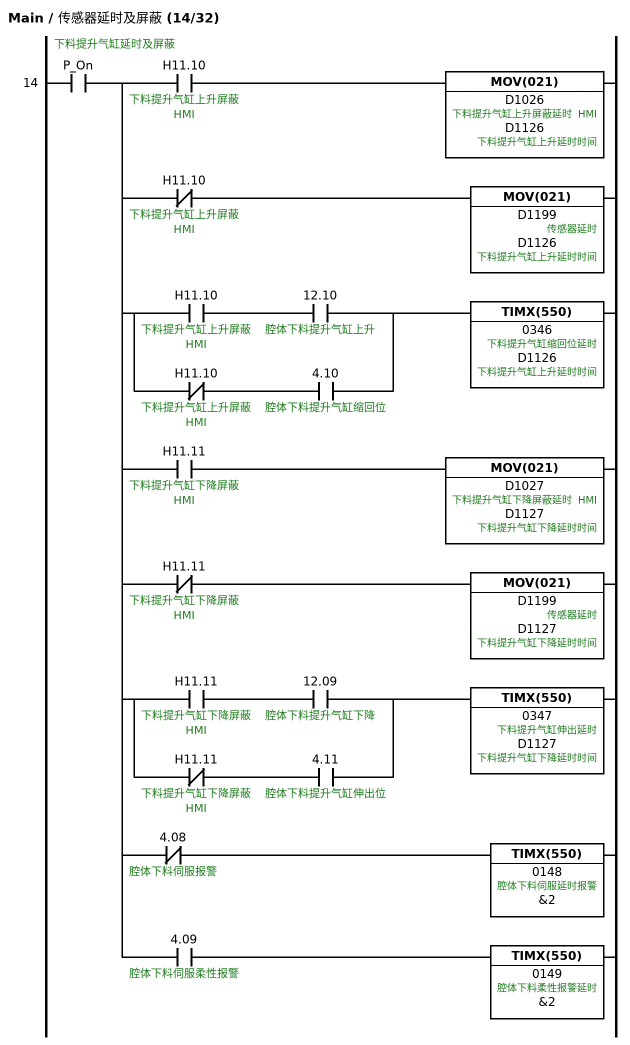
; rung 14: 下料提升气缸延时及屏蔽
LD P_On
OUT TR0
AND H11.10  ; 下料提升气缸上升屏蔽  HMI
MOV(021) D1026 D1126  ; 下料提升气缸上升屏蔽延时  HMI, 下料提升气缸上升延时时间
LD TR0
ANDNOT H11.10  ; 下料提升气缸上升屏蔽  HMI
MOV(021) D1199 D1126  ; 传感器延时, 下料提升气缸上升延时时间
LD TR0
LD H11.10  ; 下料提升气缸上升屏蔽  HMI
AND 12.10  ; 腔体下料提升气缸上升
LDNOT H11.10  ; 下料提升气缸上升屏蔽  HMI
AND 4.10  ; 腔体下料提升气缸缩回位
ORLD
ANDLD
TIMX(550) 0346 D1126  ; 下料提升气缸上升延时时间, 下料提升气缸缩回位延时
LD TR0
AND H11.11  ; 下料提升气缸下降屏蔽  HMI
MOV(021) D1027 D1127  ; 下料提升气缸下降屏蔽延时  HMI, 下料提升气缸下降延时时间
LD TR0
ANDNOT H11.11  ; 下料提升气缸下降屏蔽  HMI
MOV(021) D1199 D1127  ; 传感器延时, 下料提升气缸下降延时时间
LD TR0
LD H11.11  ; 下料提升气缸下降屏蔽  HMI
AND 12.09  ; 腔体下料提升气缸下降
LDNOT H11.11  ; 下料提升气缸下降屏蔽  HMI
AND 4.11  ; 腔体下料提升气缸伸出位
ORLD
ANDLD
TIMX(550) 0347 D1127  ; 下料提升气缸下降延时时间, 下料提升气缸伸出延时
LD TR0
ANDNOT 4.08  ; 腔体下料伺服报警
TIMX(550) 0148 &2  ; 腔体下料伺服延时报警
LD TR0
AND 4.09  ; 腔体下料伺服柔性报警
TIMX(550) 0149 &2  ; 腔体下料柔性报警延时

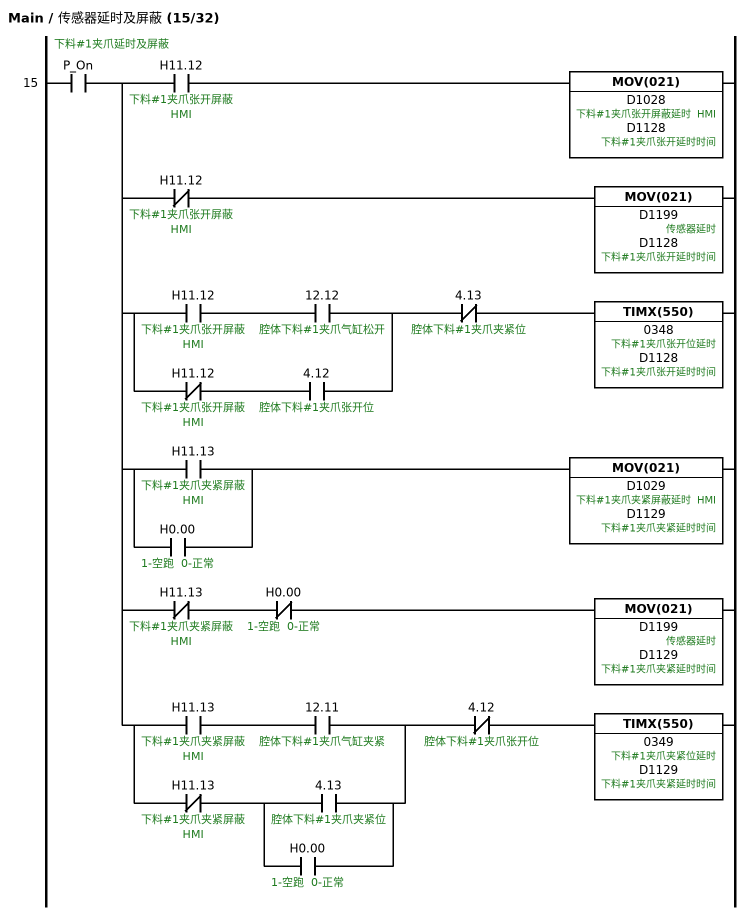
; rung 15: 下料#1夹爪延时及屏蔽
LD P_On
OUT TR0
AND H11.12  ; 下料#1夹爪张开屏蔽  HMI
MOV(021) D1028 D1128  ; 下料#1夹爪张开屏蔽延时  HMI, 下料#1夹爪张开延时时间
LD TR0
ANDNOT H11.12  ; 下料#1夹爪张开屏蔽  HMI
MOV(021) D1199 D1128  ; 传感器延时, 下料#1夹爪张开延时时间
LD TR0
LD H11.12  ; 下料#1夹爪张开屏蔽  HMI
AND 12.12  ; 腔体下料#1夹爪气缸松开
LDNOT H11.12  ; 下料#1夹爪张开屏蔽  HMI
AND 4.12  ; 腔体下料#1夹爪张开位
ORLD
ANDLD
ANDNOT 4.13  ; 腔体下料#1夹爪夹紧位
TIMX(550) 0348 D1128  ; 下料#1夹爪张开延时时间, 下料#1夹爪张开位延时
LD TR0
LD H11.13  ; 下料#1夹爪夹紧屏蔽  HMI
OR H0.00  ; 1-空跑  0-正常
ANDLD
MOV(021) D1029 D1129  ; 下料#1夹爪夹紧屏蔽延时  HMI, 下料#1夹爪夹紧延时时间
LD TR0
ANDNOT H11.13  ; 下料#1夹爪夹紧屏蔽  HMI
ANDNOT H0.00  ; 1-空跑  0-正常
MOV(021) D1199 D1129  ; 传感器延时, 下料#1夹爪夹紧延时时间
LD TR0
LD H11.13  ; 下料#1夹爪夹紧屏蔽  HMI
AND 12.11  ; 腔体下料#1夹爪气缸夹紧
LDNOT H11.13  ; 下料#1夹爪夹紧屏蔽  HMI
LD 4.13  ; 腔体下料#1夹爪夹紧位
OR H0.00  ; 1-空跑  0-正常
ANDLD
ORLD
ANDLD
ANDNOT 4.12  ; 腔体下料#1夹爪张开位
TIMX(550) 0349 D1129  ; 下料#1夹爪夹紧延时时间, 下料#1夹爪夹紧位延时

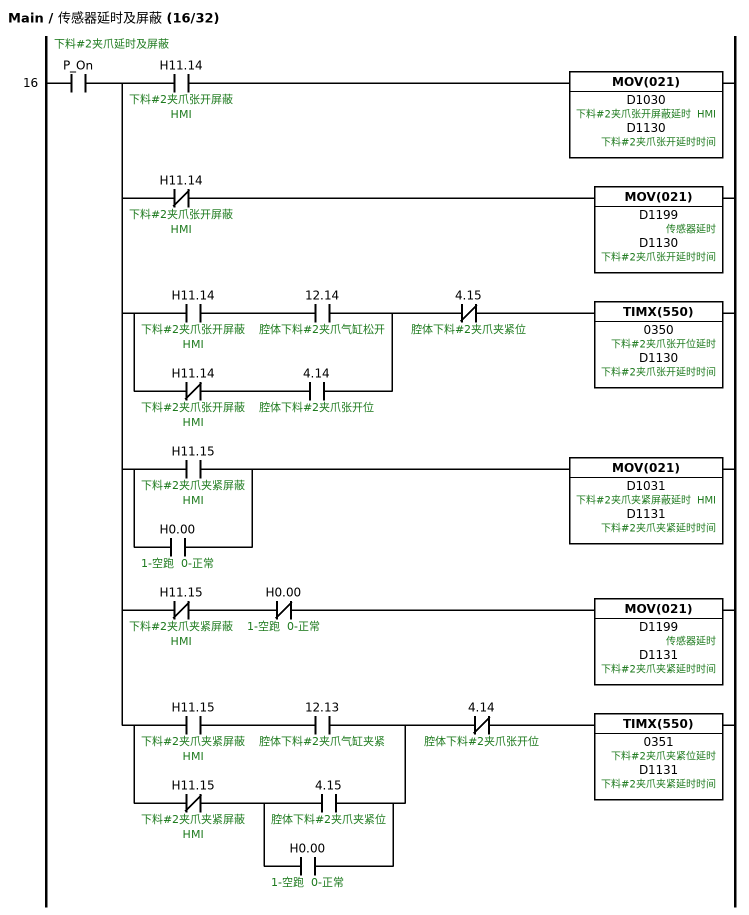
; rung 16: 下料#2夹爪延时及屏蔽
LD P_On
OUT TR0
AND H11.14  ; 下料#2夹爪张开屏蔽  HMI
MOV(021) D1030 D1130  ; 下料#2夹爪张开屏蔽延时  HMI, 下料#2夹爪张开延时时间
LD TR0
ANDNOT H11.14  ; 下料#2夹爪张开屏蔽  HMI
MOV(021) D1199 D1130  ; 传感器延时, 下料#2夹爪张开延时时间
LD TR0
LD H11.14  ; 下料#2夹爪张开屏蔽  HMI
AND 12.14  ; 腔体下料#2夹爪气缸松开
LDNOT H11.14  ; 下料#2夹爪张开屏蔽  HMI
AND 4.14  ; 腔体下料#2夹爪张开位
ORLD
ANDLD
ANDNOT 4.15  ; 腔体下料#2夹爪夹紧位
TIMX(550) 0350 D1130  ; 下料#2夹爪张开延时时间, 下料#2夹爪张开位延时
LD TR0
LD H11.15  ; 下料#2夹爪夹紧屏蔽  HMI
OR H0.00  ; 1-空跑  0-正常
ANDLD
MOV(021) D1031 D1131  ; 下料#2夹爪夹紧屏蔽延时  HMI, 下料#2夹爪夹紧延时时间
LD TR0
ANDNOT H11.15  ; 下料#2夹爪夹紧屏蔽  HMI
ANDNOT H0.00  ; 1-空跑  0-正常
MOV(021) D1199 D1131  ; 传感器延时, 下料#2夹爪夹紧延时时间
LD TR0
LD H11.15  ; 下料#2夹爪夹紧屏蔽  HMI
AND 12.13  ; 腔体下料#2夹爪气缸夹紧
LDNOT H11.15  ; 下料#2夹爪夹紧屏蔽  HMI
LD 4.15  ; 腔体下料#2夹爪夹紧位
OR H0.00  ; 1-空跑  0-正常
ANDLD
ORLD
ANDLD
ANDNOT 4.14  ; 腔体下料#2夹爪张开位
TIMX(550) 0351 D1131  ; 下料#2夹爪夹紧延时时间, 下料#2夹爪夹紧位延时

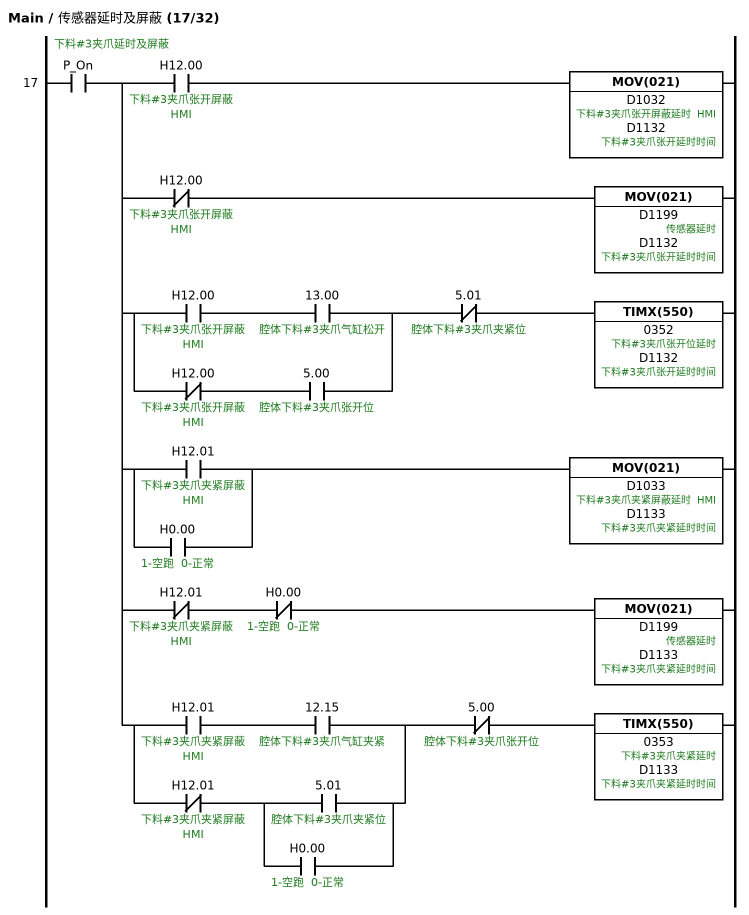
; rung 17: 下料#3夹爪延时及屏蔽
LD P_On
OUT TR0
AND H12.00  ; 下料#3夹爪张开屏蔽  HMI
MOV(021) D1032 D1132  ; 下料#3夹爪张开屏蔽延时  HMI, 下料#3夹爪张开延时时间
LD TR0
ANDNOT H12.00  ; 下料#3夹爪张开屏蔽  HMI
MOV(021) D1199 D1132  ; 传感器延时, 下料#3夹爪张开延时时间
LD TR0
LD H12.00  ; 下料#3夹爪张开屏蔽  HMI
AND 13.00  ; 腔体下料#3夹爪气缸松开
LDNOT H12.00  ; 下料#3夹爪张开屏蔽  HMI
AND 5.00  ; 腔体下料#3夹爪张开位
ORLD
ANDLD
ANDNOT 5.01  ; 腔体下料#3夹爪夹紧位
TIMX(550) 0352 D1132  ; 下料#3夹爪张开延时时间, 下料#3夹爪张开位延时
LD TR0
LD H12.01  ; 下料#3夹爪夹紧屏蔽  HMI
OR H0.00  ; 1-空跑  0-正常
ANDLD
MOV(021) D1033 D1133  ; 下料#3夹爪夹紧屏蔽延时  HMI, 下料#3夹爪夹紧延时时间
LD TR0
ANDNOT H12.01  ; 下料#3夹爪夹紧屏蔽  HMI
ANDNOT H0.00  ; 1-空跑  0-正常
MOV(021) D1199 D1133  ; 传感器延时, 下料#3夹爪夹紧延时时间
LD TR0
LD H12.01  ; 下料#3夹爪夹紧屏蔽  HMI
AND 12.15  ; 腔体下料#3夹爪气缸夹紧
LDNOT H12.01  ; 下料#3夹爪夹紧屏蔽  HMI
LD 5.01  ; 腔体下料#3夹爪夹紧位
OR H0.00  ; 1-空跑  0-正常
ANDLD
ORLD
ANDLD
ANDNOT 5.00  ; 腔体下料#3夹爪张开位
TIMX(550) 0353 D1133  ; 下料#3夹爪夹紧延时时间, 下料#3夹爪夹紧延时

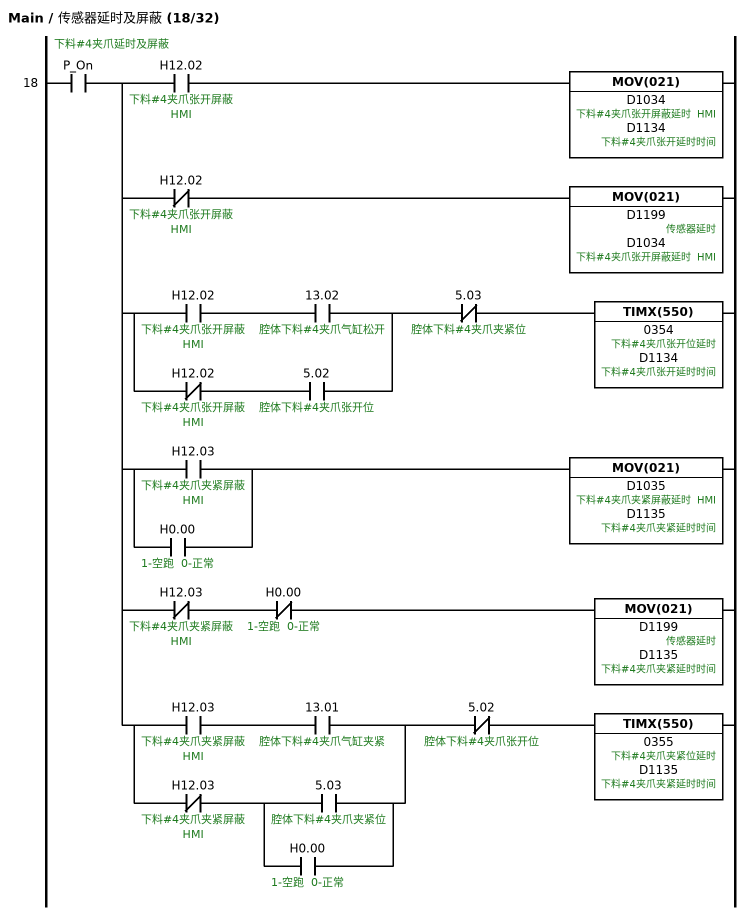
; rung 18: 下料#4夹爪延时及屏蔽
LD P_On
OUT TR0
AND H12.02  ; 下料#4夹爪张开屏蔽  HMI
MOV(021) D1034 D1134  ; 下料#4夹爪张开屏蔽延时  HMI, 下料#4夹爪张开延时时间
LD TR0
ANDNOT H12.02  ; 下料#4夹爪张开屏蔽  HMI
MOV(021) D1199 D1034  ; 传感器延时, 下料#4夹爪张开屏蔽延时  HMI
LD TR0
LD H12.02  ; 下料#4夹爪张开屏蔽  HMI
AND 13.02  ; 腔体下料#4夹爪气缸松开
LDNOT H12.02  ; 下料#4夹爪张开屏蔽  HMI
AND 5.02  ; 腔体下料#4夹爪张开位
ORLD
ANDLD
ANDNOT 5.03  ; 腔体下料#4夹爪夹紧位
TIMX(550) 0354 D1134  ; 下料#4夹爪张开延时时间, 下料#4夹爪张开位延时
LD TR0
LD H12.03  ; 下料#4夹爪夹紧屏蔽  HMI
OR H0.00  ; 1-空跑  0-正常
ANDLD
MOV(021) D1035 D1135  ; 下料#4夹爪夹紧屏蔽延时  HMI, 下料#4夹爪夹紧延时时间
LD TR0
ANDNOT H12.03  ; 下料#4夹爪夹紧屏蔽  HMI
ANDNOT H0.00  ; 1-空跑  0-正常
MOV(021) D1199 D1135  ; 传感器延时, 下料#4夹爪夹紧延时时间
LD TR0
LD H12.03  ; 下料#4夹爪夹紧屏蔽  HMI
AND 13.01  ; 腔体下料#4夹爪气缸夹紧
LDNOT H12.03  ; 下料#4夹爪夹紧屏蔽  HMI
LD 5.03  ; 腔体下料#4夹爪夹紧位
OR H0.00  ; 1-空跑  0-正常
ANDLD
ORLD
ANDLD
ANDNOT 5.02  ; 腔体下料#4夹爪张开位
TIMX(550) 0355 D1135  ; 下料#4夹爪夹紧延时时间, 下料#4夹爪夹紧位延时

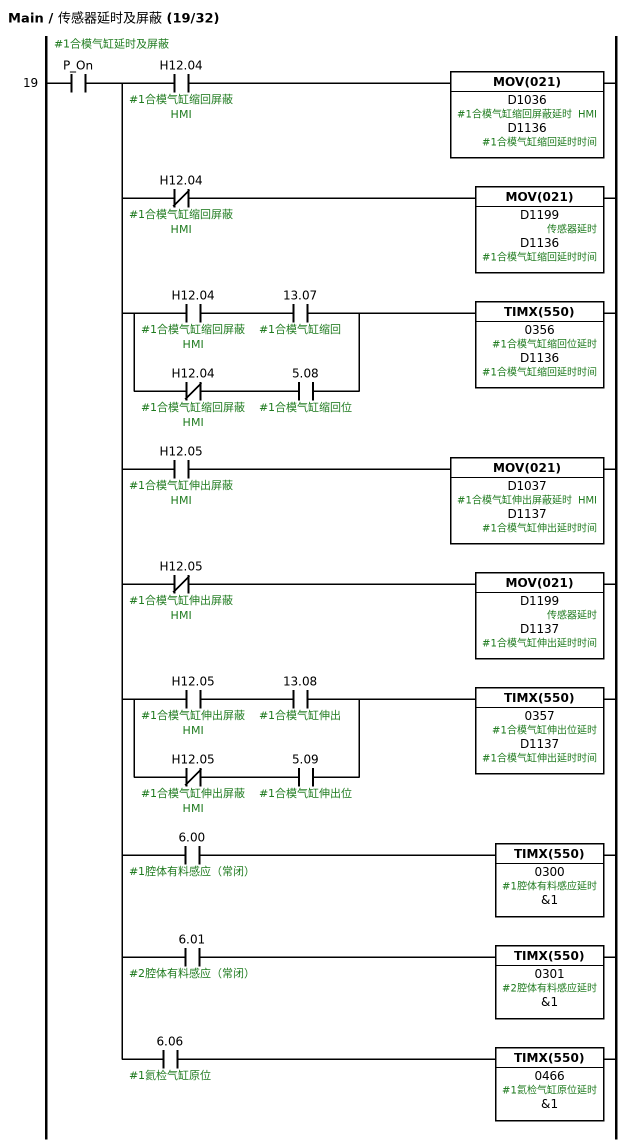
; rung 19: #1合模气缸延时及屏蔽
LD P_On
OUT TR0
AND H12.04  ; #1合模气缸缩回屏蔽  HMI
MOV(021) D1036 D1136  ; #1合模气缸缩回屏蔽延时  HMI, #1合模气缸缩回延时时间
LD TR0
ANDNOT H12.04  ; #1合模气缸缩回屏蔽  HMI
MOV(021) D1199 D1136  ; 传感器延时, #1合模气缸缩回延时时间
LD TR0
LD H12.04  ; #1合模气缸缩回屏蔽  HMI
AND 13.07  ; #1合模气缸缩回
LDNOT H12.04  ; #1合模气缸缩回屏蔽  HMI
AND 5.08  ; #1合模气缸缩回位
ORLD
ANDLD
TIMX(550) 0356 D1136  ; #1合模气缸缩回延时时间, #1合模气缸缩回位延时
LD TR0
AND H12.05  ; #1合模气缸伸出屏蔽  HMI
MOV(021) D1037 D1137  ; #1合模气缸伸出屏蔽延时  HMI, #1合模气缸伸出延时时间
LD TR0
ANDNOT H12.05  ; #1合模气缸伸出屏蔽  HMI
MOV(021) D1199 D1137  ; 传感器延时, #1合模气缸伸出延时时间
LD TR0
LD H12.05  ; #1合模气缸伸出屏蔽  HMI
AND 13.08  ; #1合模气缸伸出
LDNOT H12.05  ; #1合模气缸伸出屏蔽  HMI
AND 5.09  ; #1合模气缸伸出位
ORLD
ANDLD
TIMX(550) 0357 D1137  ; #1合模气缸伸出延时时间, #1合模气缸伸出位延时
LD TR0
AND 6.00  ; #1腔体有料感应（常闭）
TIMX(550) 0300 &1  ; #1腔体有料感应延时
LD TR0
AND 6.01  ; #2腔体有料感应（常闭）
TIMX(550) 0301 &1  ; #2腔体有料感应延时
LD TR0
AND 6.06  ; #1氦检气缸原位
TIMX(550) 0466 &1  ; #1氦检气缸原位延时

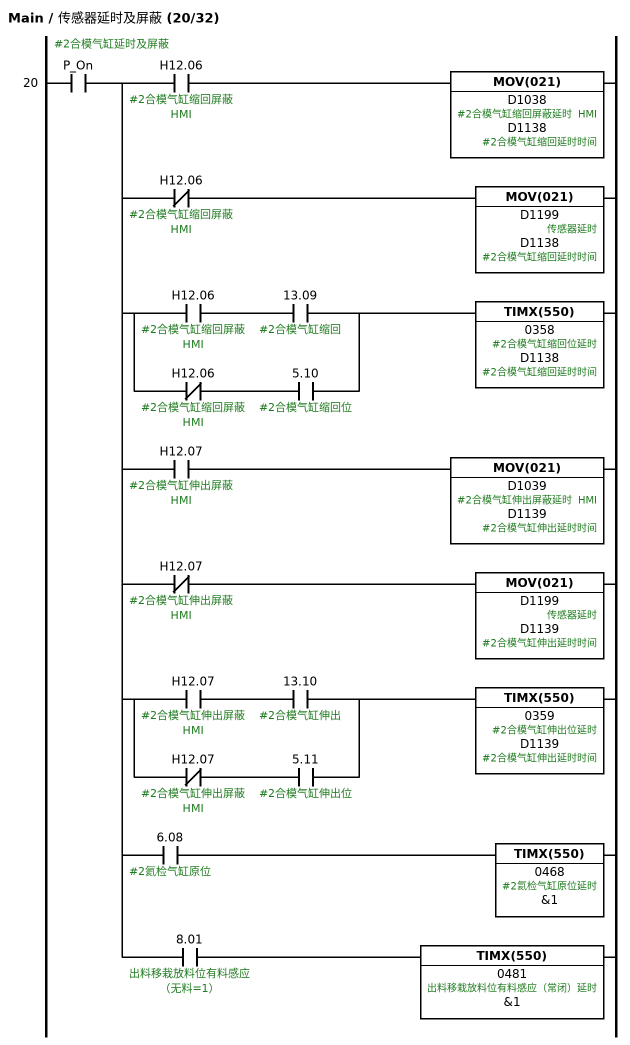
; rung 20: #2合模气缸延时及屏蔽
LD P_On
OUT TR0
AND H12.06  ; #2合模气缸缩回屏蔽  HMI
MOV(021) D1038 D1138  ; #2合模气缸缩回屏蔽延时  HMI, #2合模气缸缩回延时时间
LD TR0
ANDNOT H12.06  ; #2合模气缸缩回屏蔽  HMI
MOV(021) D1199 D1138  ; 传感器延时, #2合模气缸缩回延时时间
LD TR0
LD H12.06  ; #2合模气缸缩回屏蔽  HMI
AND 13.09  ; #2合模气缸缩回
LDNOT H12.06  ; #2合模气缸缩回屏蔽  HMI
AND 5.10  ; #2合模气缸缩回位
ORLD
ANDLD
TIMX(550) 0358 D1138  ; #2合模气缸缩回延时时间, #2合模气缸缩回位延时
LD TR0
AND H12.07  ; #2合模气缸伸出屏蔽  HMI
MOV(021) D1039 D1139  ; #2合模气缸伸出屏蔽延时  HMI, #2合模气缸伸出延时时间
LD TR0
ANDNOT H12.07  ; #2合模气缸伸出屏蔽  HMI
MOV(021) D1199 D1139  ; 传感器延时, #2合模气缸伸出延时时间
LD TR0
LD H12.07  ; #2合模气缸伸出屏蔽  HMI
AND 13.10  ; #2合模气缸伸出
LDNOT H12.07  ; #2合模气缸伸出屏蔽  HMI
AND 5.11  ; #2合模气缸伸出位
ORLD
ANDLD
TIMX(550) 0359 D1139  ; #2合模气缸伸出延时时间, #2合模气缸伸出位延时
LD TR0
AND 6.08  ; #2氦检气缸原位
TIMX(550) 0468 &1  ; #2氦检气缸原位延时
LD TR0
AND 8.01  ; 出料移栽放料位有料感应（无料=1）
TIMX(550) 0481 &1  ; 出料移栽放料位有料感应（常闭）延时

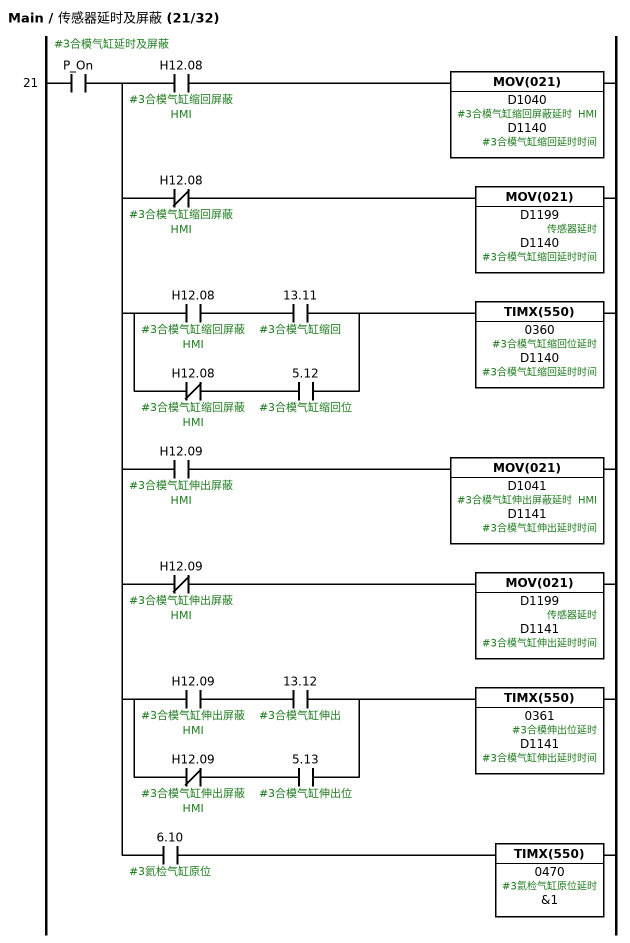
; rung 21: #3合模气缸延时及屏蔽
LD P_On
OUT TR0
AND H12.08  ; #3合模气缸缩回屏蔽  HMI
MOV(021) D1040 D1140  ; #3合模气缸缩回屏蔽延时  HMI, #3合模气缸缩回延时时间
LD TR0
ANDNOT H12.08  ; #3合模气缸缩回屏蔽  HMI
MOV(021) D1199 D1140  ; 传感器延时, #3合模气缸缩回延时时间
LD TR0
LD H12.08  ; #3合模气缸缩回屏蔽  HMI
AND 13.11  ; #3合模气缸缩回
LDNOT H12.08  ; #3合模气缸缩回屏蔽  HMI
AND 5.12  ; #3合模气缸缩回位
ORLD
ANDLD
TIMX(550) 0360 D1140  ; #3合模气缸缩回延时时间, #3合模气缸缩回位延时
LD TR0
AND H12.09  ; #3合模气缸伸出屏蔽  HMI
MOV(021) D1041 D1141  ; #3合模气缸伸出屏蔽延时  HMI, #3合模气缸伸出延时时间
LD TR0
ANDNOT H12.09  ; #3合模气缸伸出屏蔽  HMI
MOV(021) D1199 D1141  ; 传感器延时, #3合模气缸伸出延时时间
LD TR0
LD H12.09  ; #3合模气缸伸出屏蔽  HMI
AND 13.12  ; #3合模气缸伸出
LDNOT H12.09  ; #3合模气缸伸出屏蔽  HMI
AND 5.13  ; #3合模气缸伸出位
ORLD
ANDLD
TIMX(550) 0361 D1141  ; #3合模气缸伸出延时时间, #3合模伸出位延时
LD TR0
AND 6.10  ; #3氦检气缸原位
TIMX(550) 0470 &1  ; #3氦检气缸原位延时

